FUNCTION_BLOCK B_SECCOM_INFORMEFIJO (* Basic Function Block Type *)
  (* Standard: 61499-2 *)
  (* Version 0.0, 2015-11-24, 4DIAC-IDE, 4DIAC-Consortium *)
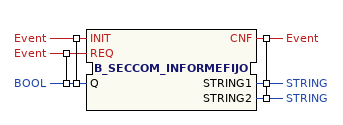
  EVENT_INPUT
    INIT WITH Q; (* Initialization Request *)
    REQ WITH Q; (* Normal Execution Request *)
  END_EVENT
  EVENT_OUTPUT
    CNF WITH STRING1, STRING2; (* Execution Confirmation *)
  END_EVENT
  VAR_INPUT
    Q : BOOL;
  END_VAR
  VAR_OUTPUT
    STRING1 : STRING;
    STRING2 : STRING;
  END_VAR
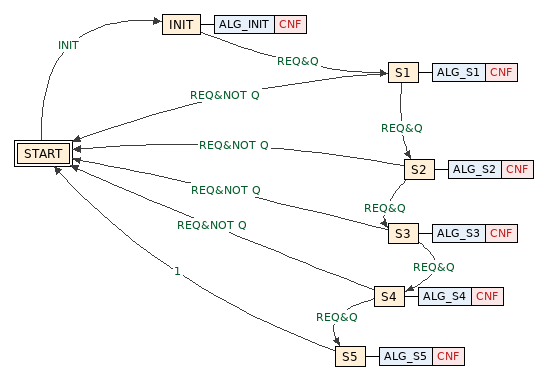
  EC_STATES
    START; (* Initial State *)
    INIT : ALG_INIT -> CNF; (* Initialization *)
    S1 : ALG_S1 -> CNF;
    S2 : ALG_S2 -> CNF;
    S3 : ALG_S3 -> CNF;
    S4 : ALG_S4 -> CNF;
    S5 : ALG_S5 -> CNF;
  END_STATES
  EC_TRANSITIONS
    START TO INIT := INIT;
    INIT TO S1 := REQ&Q;
    S1 TO START := REQ&NOT Q;
    S1 TO S2 := REQ&Q;
    S2 TO START := REQ&NOT Q;
    S2 TO S3 := REQ&Q;
    S3 TO START := REQ&NOT Q;
    S3 TO S4 := REQ&Q;
    S4 TO START := REQ&NOT Q;
    S4 TO S5 := REQ&Q;
    S5 TO START := 1;
  END_TRANSITIONS
  ALGORITHM ALG_INIT IN ST: (* new algorithm *)
STRING1:='\x04\x7f';
STRING2:='\x01\x02\x03\x04';
  END_ALGORITHM
  ALGORITHM ALG_S1 IN ST: (* new algorithm *)
STRING1:='\x05';
STRING2:='\x10\x30';
  END_ALGORITHM
  ALGORITHM ALG_S2 IN ST: (* new algorithm *)
STRING1:='\x01\x52\x43\x4c\x02\x03\xfe\x2c';
STRING2:='\x10\x31';
  END_ALGORITHM
  ALGORITHM ALG_S3 IN ST: (* new algorithm *)
STRING1:='\x04';
STRING2:='\x05\x7f';
  END_ALGORITHM
  ALGORITHM ALG_S4 IN ST: (* new algorithm *)
STRING1:='\x10\x30';
STRING2:='\x02\x03';
  END_ALGORITHM
  ALGORITHM ALG_S5 IN ST: (* new algorithm *)
STRING1:='\x10\x31';
STRING2:='\x04\x7f';
  END_ALGORITHM
END_FUNCTION_BLOCK
